(*
Nazwa:			FB_InputFilter
Opis: 			Filtrowanie czujnikow
Wersja:			v1.0
Data:			2023-09-20
Autor:			DP
Urzadzenia:		
Konfiguracja:	
Info:
- blok filtrujacy wejście cyfrowe
*)

FUNCTION_BLOCK FB_InputFilter
VAR_INPUT
	bIN:BOOL;				//Wejście cyfrowe
	tFilterTimeOn:TIME;		//Czas filtrowania
	tFilterTimeOff:TIME;	//Czas filtrowania
END_VAR
VAR_OUTPUT
	bOUT:BOOL;
END_VAR
VAR
	tonIN: TON;
	tonOFF: TOF;
END_VAR


(* w1
tonOFF(IN:=bIN, PT:=tFilterTimeOff);
tonIN(IN:=tonOFF.Q, PT:=tFilterTimeOn);
bOUT:=tonIN.Q;
*)

(* w2 *)
tonIN	(IN:=bIN, 		PT:=tFilterTimeOn);
tonOFF	(IN:=NOT bIN, 	PT:=tFilterTimeOff);
IF tonIN.Q THEN
	bOUT := 	TRUE;
ELSIF tonOFF.Q THEN
	bOUT := 	FALSE;
END_IF

END_FUNCTION_BLOCK

(* stored: Version 1.1.0.1, ProductVersion 3.1.4026.13, FileIdentifier 19a61f5727d774f54514f475db9431e5bae95001, FileSignature 224a9dc8abb7f794cb2af57d1223c82367966df5d64b44bca252b050adc750b3fb43fb981468b8339499d2f0054a10fa576940fdefeb166300c38a2ac89d3e010aab2ff2098fb4e3e7b0497ba43ebea641769e0e844a581de60c32112186f998f5b25d04c2d33e507a097b323cb24d661ce455e2b45039dc2def7cb31d53f54ea18b8a7db7b2eec1d0543235b6c20b1a2b23e916d62468b01ffd606e4e1a3ca9570fa0b1fbf52f6aade486230587e9b6e58ff6eefaf28b9a6f1323fad167ca3b316dc4173870512efb302520ea09f515b7ab6fe7a0effbfd31453810ac6bb19f1e5f3f2fef842c6f41bd87e93a313979361b912ec7a95b97f3a0c390245285af
   POU FB_InputFilter: Id {15a70139-ebba-4342-b522-5592b8dff86d}, SpecialFunc None *)
